{attribute 'pack_mode' := '1'}//Ensures 1-byte-alignmend
TYPE AX5000_P_0206 :
STRUCT
	Actual_lenght:UINT;
	Max_lenght:UINT;
	Umain_max_critical_hardware_voltage:UINT;
	Umain_min_critical_hardware_voltage:UINT;
	Umain_overvoltage_threshold:UINT;
	Umain_underervoltage_threshold:UINT;
	Umain_peak_overvoltage_threshold:UINT;
	Umain_peak_underervoltage_threshold:UINT;
	Umain_peak_lost_phase_threshold:UINT;
	Internal_brake_chopper_on_threshold:UINT;
	Internal_brake_chopper_off_threshold:UINT;
	Base_internal_brake_chopper_on_threshold:UINT;
	External_brake_chopper_on_threshold:UINT;
	External_brake_chopper_off_threshold:UINT;
	Base_external_brake_chopper_on_threshold:UINT;
	External_dc_link_connection_off_threshold:UINT;
	DCLink_volervoltage_on_threshold:UINT;
	DCLink_undervoltage_off_threshold:UINT;
	DCLink_undervoltage_warning_threshold:UINT;
	DCLink_undervoltage_error_threshold:UINT;
	DCLink_bypass_load_resistor_on_threshold:UINT;
	DCLink_bypass_load_resistor_off_threshold:UINT;
	External_Umain_rekay_off_threshold:UINT;
	External_Umain_rekay_on_threshold:UINT;
	AX5160_AX5193_Umain_peak_phase_monitoring_threshold:UINT;
//	{attribute 'hide'}
	Rsvd:ARRAY[0..6] OF UINT;

END_STRUCT
END_TYPE

(* stored: Version 1.1.0.1, ProductVersion 3.1.4024.4
   DUT AX5000_P_0206: Id {646ef8a3-3b98-491d-9eca-9f1b24bbe7fc} *)
